// TIA Portal V19 export
ORGANIZATION_BLOCK "Main"   // OB1, LAD, ProgramCycle
TITLE = "Main Program Sweep (Cycle)"
{ S7_Optimized_Access := 'TRUE' }
// stored: SetENOAutomatically false
   VAR_INPUT
      Initial_Call : Bool;   // Initial call of this OB
      Remanence : Bool;   // =True, if remanent data are available
   END_VAR
BEGIN

REGION Network 1: Sensor 1 - Alarm
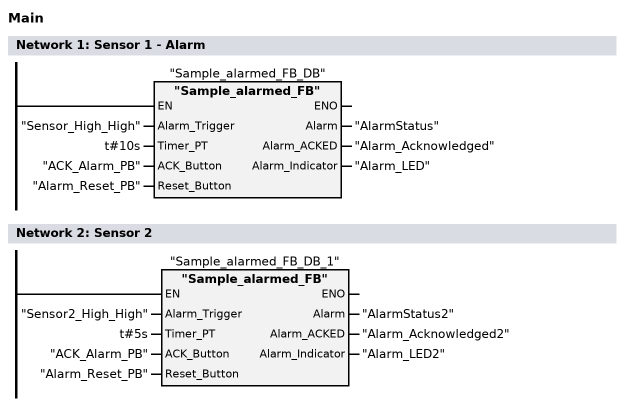
   RUNG wire#powerrail
      "Sample_alarmed_FB_DB"(Alarm_Trigger := "Sensor_High_High", Timer_PT := t#10s, ACK_Button := "ACK_Alarm_PB", Reset_Button := "Alarm_Reset_PB", Alarm => "AlarmStatus", Alarm_ACKED => "Alarm_Acknowledged", Alarm_Indicator => "Alarm_LED")
   END_RUNG
   // the same network as SCL:
   "Sample_alarmed_FB_DB"(Alarm_Trigger := "Sensor_High_High",   // "Sample_alarmed_FB"
                          Timer_PT := t#10s,
                          ACK_Button := "ACK_Alarm_PB",
                          Reset_Button := "Alarm_Reset_PB",
                          Alarm => "AlarmStatus",
                          Alarm_ACKED => "Alarm_Acknowledged",
                          Alarm_Indicator => "Alarm_LED");
END_REGION

REGION Network 2: Sensor 2
   RUNG wire#powerrail
      "Sample_alarmed_FB_DB_1"(Alarm_Trigger := "Sensor2_High_High", Timer_PT := t#5s, ACK_Button := "ACK_Alarm_PB", Reset_Button := "Alarm_Reset_PB", Alarm => "AlarmStatus2", Alarm_ACKED => "Alarm_Acknowledged2", Alarm_Indicator => "Alarm_LED2")
   END_RUNG
   // the same network as SCL:
   "Sample_alarmed_FB_DB_1"(Alarm_Trigger := "Sensor2_High_High",   // "Sample_alarmed_FB"
                           Timer_PT := t#5s,
                           ACK_Button := "ACK_Alarm_PB",
                           Reset_Button := "Alarm_Reset_PB",
                           Alarm => "AlarmStatus2",
                           Alarm_ACKED => "Alarm_Acknowledged2",
                           Alarm_Indicator => "Alarm_LED2");
END_REGION
END_ORGANIZATION_BLOCK
